// TIA Portal V17 export
// export: Created 2024-09-02T12:50:06.39653Z, ExportSetting WithDefaults, DisplayName Totally Integrated Automation Portal, DisplayVersion V17, DisplayName TIA Portal Openness, DisplayVersion V17, DisplayName TIA Portal Version Control Interface, DisplayVersion V17, DisplayName STEP 7 Professional, DisplayVersion V17, DisplayName STEP 7 Safety, DisplayVersion V17, DisplayName WinCC Professional, DisplayVersion V17
FUNCTION_BLOCK "GraFB1_FG01_Transport_OP70"   // FB1281, GRAPH
VERSION : 0.1
// stored: AcknowledgeErrorsRequired false, AutoNumber false, GraphVersion 4.0, InitialValuesAcquisition true, IsIECCheckEnabled false, LanguageInNetworks LAD, LockOperatingMode false, PermanentILProcessingInMANMode true, SetENOAutomatically false, SkipSteps false, UDAEnableTagReadback false, WithAlarmHandling true
   // inherited from GRAPH_BASE
   VAR
      OFF_SQ_BASE : Bool;
   END_VAR
   VAR_INPUT
      OFF_SQ { ExternalWritable := 'False'} : Bool := false;   // Kette ausschalten
      INIT_SQ { ExternalWritable := 'False'} : Bool := false;   // Kette in Initialzustand versetzen
      ACK_EF { ExternalWritable := 'False'} : Bool := false;   // Alle Fehler und Störungen quittieren
      S_PREV { ExternalWritable := 'False'} : Bool := false;   // Vorherigen Schritt am Parameter S_NO ausgeben
      S_NEXT { ExternalWritable := 'False'} : Bool := false;   // Nächsten Schritt am Parameter S_NO anzeigen
      SW_AUTO { ExternalWritable := 'False'} : Bool := false;   // Automtischer Betrieb
      SW_TAP { ExternalWritable := 'False'} : Bool := false;   // Halbautomatisch/Weiterschalten mit Transition
      SW_TOP { ExternalWritable := 'False'} : Bool := false;   // Halbautomatisch/Ignoriere Transition
      SW_MAN { ExternalWritable := 'False'} : Bool := false;   // Handbetrieb
      S_SEL { ExternalWritable := 'False'} : Int := 0;   // Schritt auswählen, der an S_NO ausgegeben werden soll
      S_ON { ExternalWritable := 'False'} : Bool := false;   // Schritt aktivieren, der an Parameter S_NO anliegt
      S_OFF { ExternalWritable := 'False'} : Bool := false;   // Schritt deaktivieren, der an Parameter S_NO anliegt
      T_PUSH { ExternalWritable := 'False'} : Bool := false;   // Schaltfreigabe für Transition im halbautomatischen Betrieb
   END_VAR
   VAR_OUTPUT
      S_NO { ExternalWritable := 'False'} : Int := 0;   // Schrittnummer
      S_MORE { ExternalWritable := 'False'} : Bool := false;   // Weitere Schritte sind vorhanden und können in S_NO angezeigt werden.
      S_ACTIVE { ExternalWritable := 'False'} : Bool := false;   // Schritt, der an Parameter S_NO angezeigt wird, ist aktiv
      ERR_FLT { ExternalWritable := 'False'} : Bool := false;   // Sammelfehler Interlock oder Supervision
      AUTO_ON { ExternalWritable := 'False'} : Bool := false;   // Automatischer Betrieb eingeschaltet
      TAP_ON { ExternalWritable := 'False'} : Bool := false;   // Halbautomatischer Betrieb/Schritt mit Transition eingeschaltet
      TOP_ON { ExternalWritable := 'False'} : Bool := false;   // Halbautomatischer Betrieb/Ignoriere Transition eingeschaltet
      MAN_ON { ExternalWritable := 'False'} : Bool := false;   // Handbetrieb eingeschaltet
   END_VAR
   VAR
      extBlock { S7_SetPoint := 'True'} : "LTLL_ManualGraphExt";
   END_VAR
BEGIN
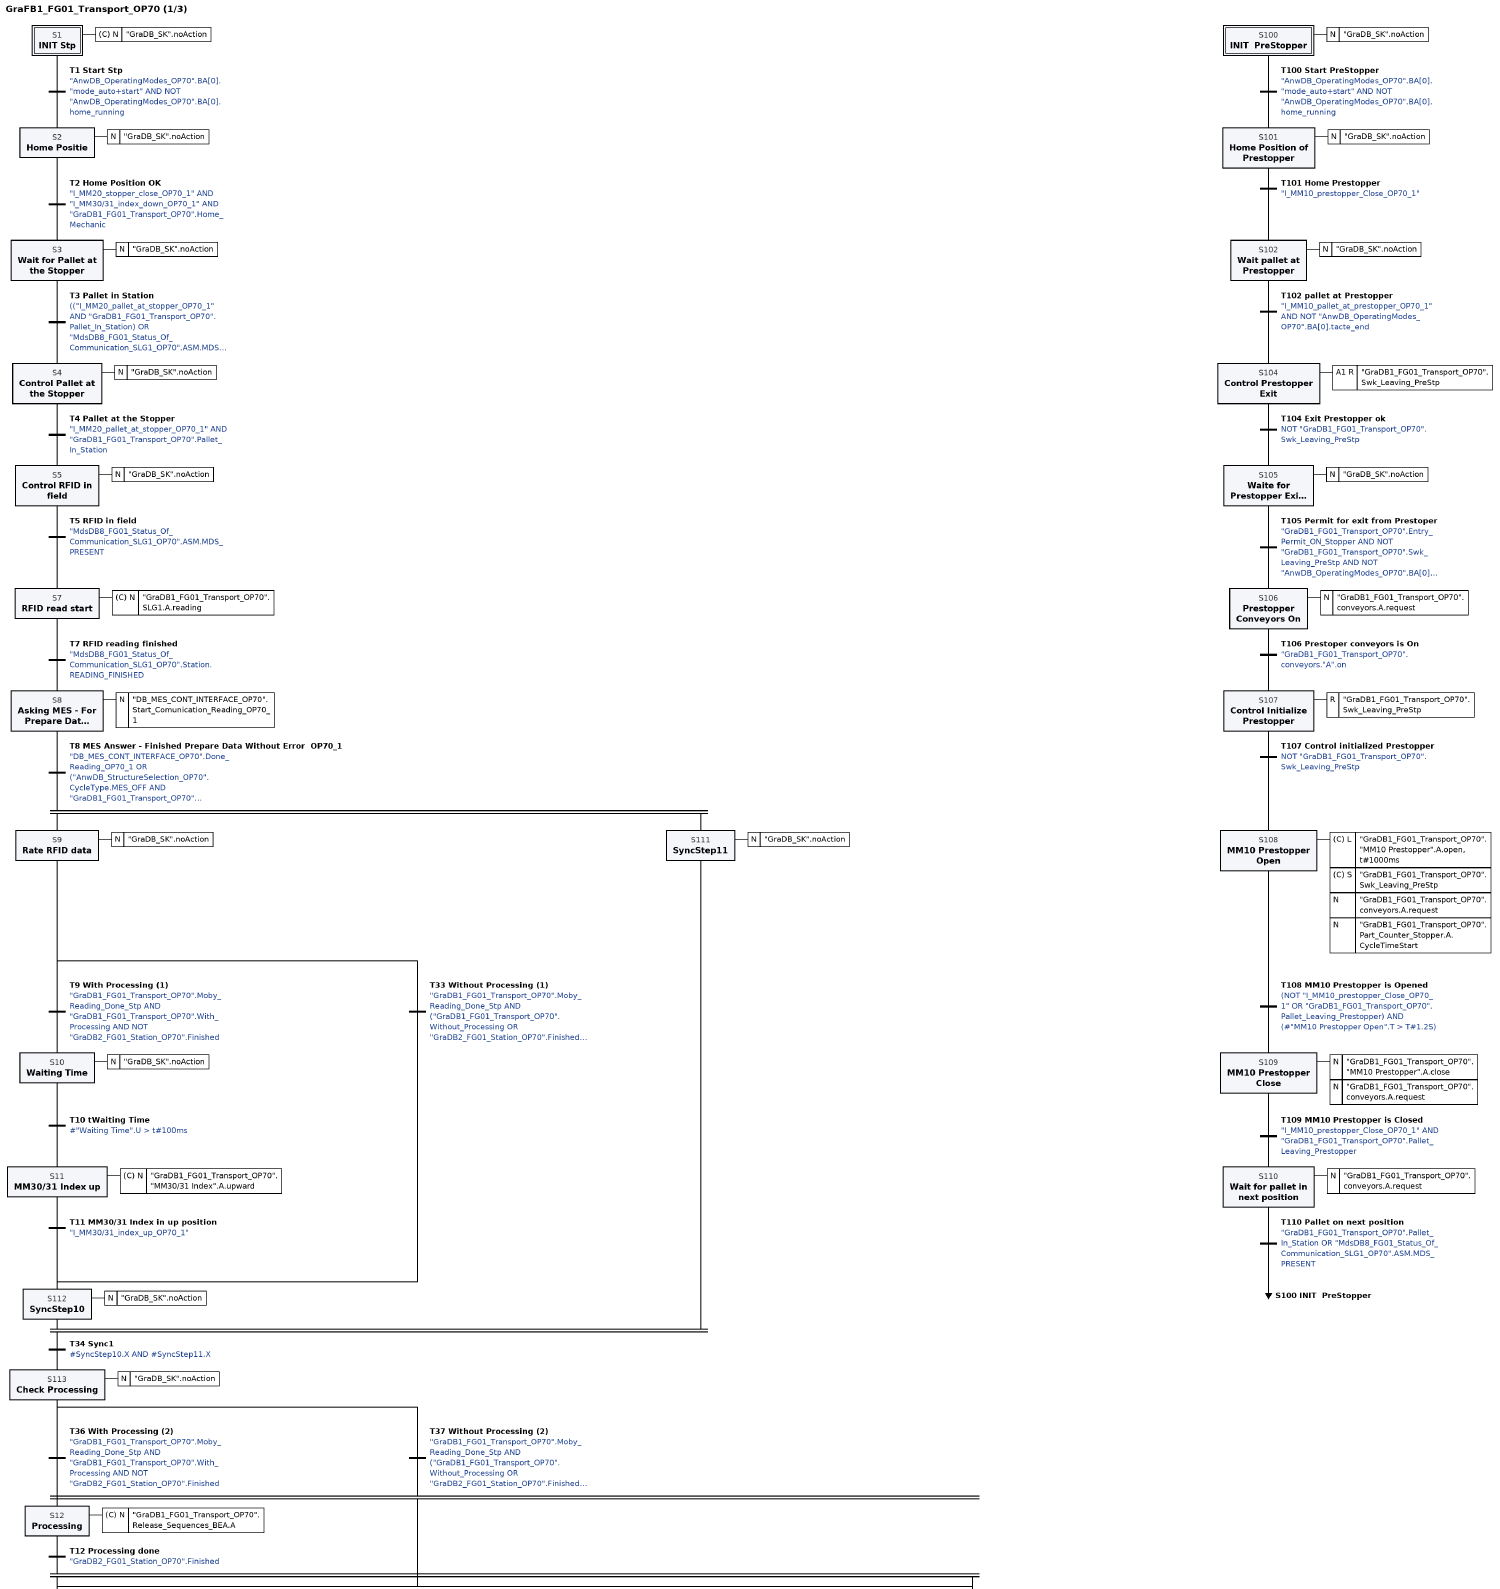
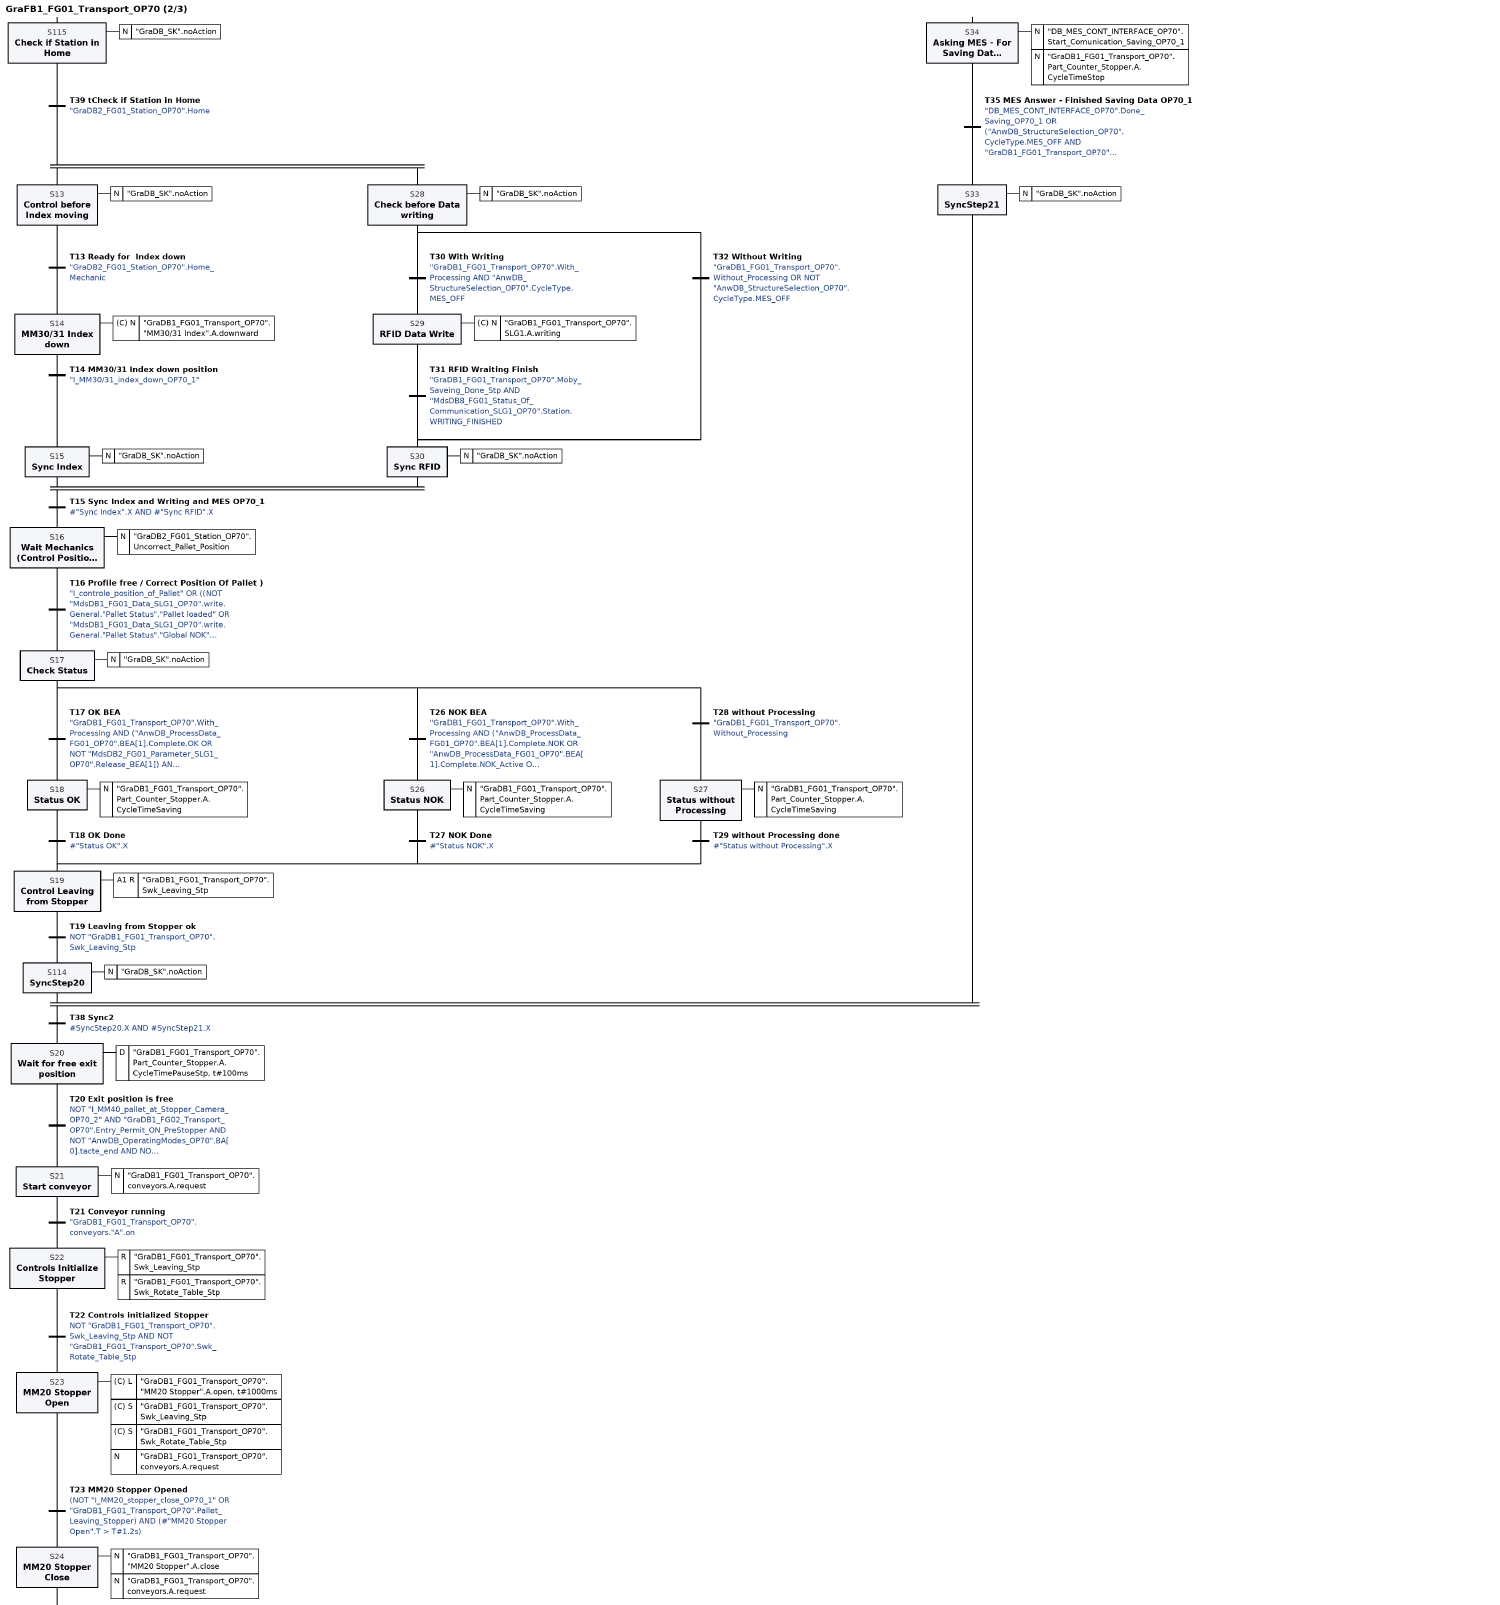
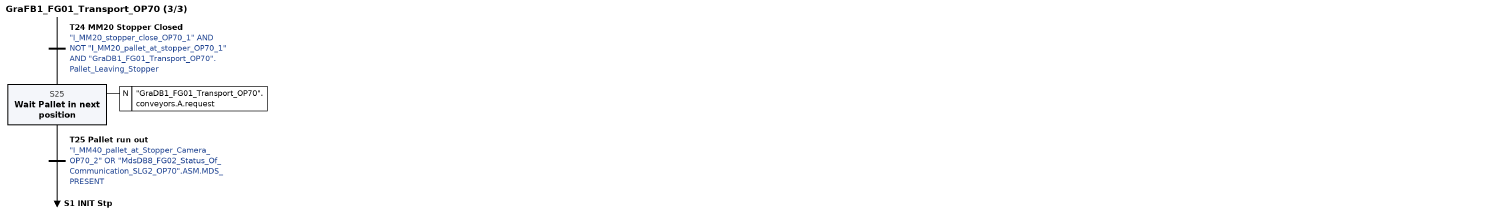
   // permanent pre-instructions
   NETWORK 1
   TITLE = HMI Lite Pass on data / HMI Lite Daten weiterreichen
      #extBlock.input := "LTLL_ManualGraphControl_OP70".screen[0].input;
   NETWORK 2
   TITLE = Instance DB Name query and pass on / Instanz DB Name abfragen und weiterreichen
      GetInstanceName(size := 0, OUT => #extBlock.input.instanceName);
   NETWORK 3
   TITLE = SK Mode
      "SysFC_SQ_Mode"(iFKT := 0, iTmsHalt := false, ioMOP := #RT_DATA.MOP);
   NETWORK 4
   TITLE = Signal change between pre-stopper and stopper / Signalwechsel Vorstopper/Stopper
      IF "GraDB1_FG01_Transport_OP70".Pallet_In_Station THEN
          "GraDB1_FG01_Transport_OP70".Swk_Leaving_PreStp := FALSE;
      END_IF;
      IF "I_MM40_pallet_at_Stopper_Camera_OP70_2" OR (NOT "GraDB1_FG01_Transport_OP70".Pallet_In_Station AND NOT "MdsDB8_FG01_Status_Of_Communication_SLG1_OP70".ASM.MDS_PRESENT AND NOT "I_MM20_pallet_at_stopper_OP70_1" AND "AlwaysFALSE") THEN
          "GraDB1_FG01_Transport_OP70".Swk_Leaving_Stp := FALSE;
      END_IF;
      IF "AlwaysTRUE" THEN "GraDB1_FG01_Transport_OP70".Swk_Rotate_Table_Stp := FALSE; END_IF;

   // sequencer 1: FG01 - Stopper MM20 / FG01 - Stopper
   INITIAL_STEP "INIT Stp":   // S1, max time T#10S, warning time T#7S
      interlock C := (none);   // Initialschritt / initial step
      supervision V := (none);   // Initialschritt / initial step
      (C)     N    "GraDB_SK".noAction
   END_STEP
   TRANSITION "Start Stp" FROM "INIT Stp" TO "Home Positie"   // T1
      := "AnwDB_OperatingModes_OP70".BA[0]."mode_auto+start" AND NOT "AnwDB_OperatingModes_OP70".BA[0].home_running;
   END_TRANSITION
   STEP "Home Positie":   // S2, max time T#10S, warning time T#7S
      supervision V := NOT #"Home Position OK".TT AND (#"Home Positie".U > T#1S);
              N    "GraDB_SK".noAction
   END_STEP
   TRANSITION "Home Position OK" FROM "Home Positie" TO "Wait for Pallet at the Stopper"   // T2
      := "I_MM20_stopper_close_OP70_1" AND "I_MM30/31_index_down_OP70_1" AND "GraDB1_FG01_Transport_OP70".Home_Mechanic;
   END_TRANSITION
   STEP "Wait for Pallet at the Stopper":   // S3, max time T#10S, warning time T#7S
              N    "GraDB_SK".noAction
   END_STEP
   TRANSITION "Pallet in Station" FROM "Wait for Pallet at the Stopper" TO "Control Pallet at the Stopper"   // T3
      := (("I_MM20_pallet_at_stopper_OP70_1" AND "GraDB1_FG01_Transport_OP70".Pallet_In_Station) OR "MdsDB8_FG01_Status_Of_Communication_SLG1_OP70".ASM.MDS_PRESENT) AND NOT "AnwDB_OperatingModes_OP70".BA[0].tacte_end;
   END_TRANSITION
   STEP "Control Pallet at the Stopper":   // S4, max time T#10S, warning time T#7S
      supervision V := NOT #"Pallet at the Stopper".TT AND (#"Control Pallet at the Stopper".U > T#5000mS);
              N    "GraDB_SK".noAction
   END_STEP
   TRANSITION "Pallet at the Stopper" FROM "Control Pallet at the Stopper" TO "Control RFID in field"   // T4
      := "I_MM20_pallet_at_stopper_OP70_1" AND "GraDB1_FG01_Transport_OP70".Pallet_In_Station;
   END_TRANSITION
   STEP "Rate RFID data":   // S9, max time T#10S, warning time T#7S
      interlock C := "MdsDB8_FG01_Status_Of_Communication_SLG1_OP70".Station.READING_FINISHED;
      supervision V := NOT #"With Processing (1)".TT AND NOT #"Without Processing (1)".TT AND (#"Rate RFID data".U > T#5000mS);
              N    "GraDB_SK".noAction
   END_STEP
   TRANSITION "With Processing (1)" FROM "Rate RFID data" TO "Waiting Time"   // T9
      := "GraDB1_FG01_Transport_OP70".Moby_Reading_Done_Stp AND "GraDB1_FG01_Transport_OP70".With_Processing AND NOT "GraDB2_FG01_Station_OP70".Finished;
   END_TRANSITION
   TRANSITION "Without Processing (1)" FROM "Rate RFID data" TO SyncStep10   // T33
      := "GraDB1_FG01_Transport_OP70".Moby_Reading_Done_Stp AND ("GraDB1_FG01_Transport_OP70".Without_Processing OR "GraDB2_FG01_Station_OP70".Finished) AND (#"Rate RFID data".T > T#500ms);
   END_TRANSITION
   STEP "MM30/31 Index up":   // S11, max time T#10S, warning time T#7S
      interlock C := "I_MM130_Press_Damper_UP_OP70_1";
      supervision V := NOT #"MM30/31 Index in up position".TT AND (#"MM30/31 Index up".U > T#5000mS);
      (C)     N    "GraDB1_FG01_Transport_OP70"."MM30/31 Index".A.upward
   END_STEP
   TRANSITION "MM30/31 Index in up position" FROM "MM30/31 Index up" TO SyncStep10   // T11
      := "I_MM30/31_index_up_OP70_1";
   END_TRANSITION
   STEP Processing:   // S12, max time T#10S, warning time T#7S
      interlock C := "MdsDB8_FG01_Status_Of_Communication_SLG1_OP70".Station.READING_FINISHED AND "I_MM30/31_index_up_OP70_1";
      (C)     N    "GraDB1_FG01_Transport_OP70".Release_Sequences_BEA.A
   END_STEP
   TRANSITION "Processing done" FROM Processing TO ("Check if Station in Home", "Asking MES - For Saving Data OP70_1")   // T12
      := "GraDB2_FG01_Station_OP70".Finished;
   END_TRANSITION
   STEP "Control before Index moving":   // S13, max time T#10S, warning time T#7S
      interlock C := "AlwaysTRUE";
      supervision V := NOT #"Ready for  Index down".TT AND (#"Control before Index moving".U > T#5000MS);
              N    "GraDB_SK".noAction
   END_STEP
   TRANSITION "Ready for  Index down" FROM "Control before Index moving" TO "MM30/31 Index  down"   // T13
      := "GraDB2_FG01_Station_OP70".Home_Mechanic;
   END_TRANSITION
   STEP "MM30/31 Index  down":   // S14, max time T#10S, warning time T#7S
      interlock C := "I_MM130_Press_Damper_UP_OP70_1";
      supervision V := NOT #"MM30/31 Index down position".TT AND (#"MM30/31 Index  down".U > T#5000mS);
      (C)     N    "GraDB1_FG01_Transport_OP70"."MM30/31 Index".A.downward
   END_STEP
   TRANSITION "MM30/31 Index down position" FROM "MM30/31 Index  down" TO "Sync Index"   // T14
      := "I_MM30/31_index_down_OP70_1";
   END_TRANSITION
   STEP "Sync Index":   // S15, max time T#10S, warning time T#7S
              N    "GraDB_SK".noAction
   END_STEP
   STEP "Check before Data writing":   // S28, max time T#10S, warning time T#7S
              N    "GraDB_SK".noAction
   END_STEP
   TRANSITION "With Writing" FROM "Check before Data writing" TO "RFID Data Write"   // T30
      := "GraDB1_FG01_Transport_OP70".With_Processing AND "AnwDB_StructureSelection_OP70".CycleType.MES_OFF;
   END_TRANSITION
   TRANSITION "Without Writing" FROM "Check before Data writing" TO "Sync RFID"   // T32
      := "GraDB1_FG01_Transport_OP70".Without_Processing OR NOT "AnwDB_StructureSelection_OP70".CycleType.MES_OFF;
   END_TRANSITION
   STEP "RFID Data Write":   // S29, max time T#10S, warning time T#7S
      interlock C := "GraDB1_FG01_Transport_OP70".Moby_Reading_Done_Stp;
      supervision V := NOT #"RFID Wraiting Finish".TT AND (#"RFID Data Write".U > T#5000MS);
      (C)     N    "GraDB1_FG01_Transport_OP70".SLG1.A.writing
   END_STEP
   TRANSITION "RFID Wraiting Finish" FROM "RFID Data Write" TO "Sync RFID"   // T31
      := "GraDB1_FG01_Transport_OP70".Moby_Saveing_Done_Stp AND "MdsDB8_FG01_Status_Of_Communication_SLG1_OP70".Station.WRITING_FINISHED;
   END_TRANSITION
   STEP "Sync RFID":   // S30, max time T#10S, warning time T#7S
              N    "GraDB_SK".noAction
   END_STEP
   TRANSITION "Sync Index and Writing and MES OP70_1" FROM ("Sync Index", "Sync RFID") TO "Wait Mechanics (Control Position Of Pallet )"   // T15
      := #"Sync Index".X AND #"Sync RFID".X;
   END_TRANSITION
   STEP "Wait Mechanics (Control Position Of Pallet )":   // S16, max time T#10S, warning time T#7S
      supervision V := NOT #"Profile free / Correct Position Of Pallet )".TT AND (#"Wait Mechanics (Control Position Of Pallet )".U > T#1000mS);
              N    "GraDB2_FG01_Station_OP70".Uncorrect_Pallet_Position
   END_STEP
   TRANSITION "Profile free / Correct Position Of Pallet )" FROM "Wait Mechanics (Control Position Of Pallet )" TO "Check Status"   // T16
      := "I_controle_position_of_Pallet" OR ((NOT "MdsDB1_FG01_Data_SLG1_OP70".write.General."Pallet Status"."Pallet loaded" OR "MdsDB1_FG01_Data_SLG1_OP70".write.General."Pallet Status"."Global NOK") AND "AnwDB_StructureSelection_OP70".CycleType.MES_OFF) OR (("DBi_Aveva_OP70_1".SettingSpecyfications.Global.General_Info.ProductStatus = 3) AND NOT "AnwDB_StructureSelection_OP70".CycleType.MES_OFF);
   END_TRANSITION
   STEP "Check Status":   // S17, max time T#10S, warning time T#7S
      supervision V := NOT #"OK BEA".TT AND NOT #"OK BEA".TT AND NOT #"without Processing".TT AND (#"Check Status".U > T#1000MS);
              N    "GraDB_SK".noAction
   END_STEP
   TRANSITION "OK BEA" FROM "Check Status" TO "Status OK"   // T17
      := "GraDB1_FG01_Transport_OP70".With_Processing AND ("AnwDB_ProcessData_FG01_OP70".BEA[1].Complete.OK OR NOT "MdsDB2_FG01_Parameter_SLG1_OP70".Release_BEA[1]) AND ("AnwDB_ProcessData_FG01_OP70".BEA[2].Complete.OK OR NOT "MdsDB2_FG01_Parameter_SLG1_OP70".Release_BEA[2]);
   END_TRANSITION
   TRANSITION "NOK BEA" FROM "Check Status" TO "Status NOK"   // T26
      := "GraDB1_FG01_Transport_OP70".With_Processing AND ("AnwDB_ProcessData_FG01_OP70".BEA[1].Complete.NOK OR "AnwDB_ProcessData_FG01_OP70".BEA[1].Complete.NOK_Active OR "AnwDB_ProcessData_FG01_OP70".BEA[2].Complete.NOK OR "AnwDB_ProcessData_FG01_OP70".BEA[2].Complete.NOK_Active);
   END_TRANSITION
   TRANSITION "without Processing" FROM "Check Status" TO "Status without Processing"   // T28
      := "GraDB1_FG01_Transport_OP70".Without_Processing;
   END_TRANSITION
   STEP "Status OK":   // S18, max time T#10S, warning time T#7S
              N    "GraDB1_FG01_Transport_OP70".Part_Counter_Stopper.A.CycleTimeSaving
   END_STEP
   TRANSITION "OK Done" FROM "Status OK" TO "Control Leaving from Stopper"   // T18
      := #"Status OK".X;
   END_TRANSITION
   STEP "Status NOK":   // S26, max time T#10S, warning time T#7S
              N    "GraDB1_FG01_Transport_OP70".Part_Counter_Stopper.A.CycleTimeSaving
   END_STEP
   TRANSITION "NOK Done" FROM "Status NOK" TO "Control Leaving from Stopper"   // T27
      := #"Status NOK".X;
   END_TRANSITION
   STEP "Status without Processing":   // S27, max time T#10S, warning time T#7S
              N    "GraDB1_FG01_Transport_OP70".Part_Counter_Stopper.A.CycleTimeSaving
   END_STEP
   TRANSITION "without Processing done" FROM "Status without Processing" TO "Control Leaving from Stopper"   // T29
      := #"Status without Processing".X;
   END_TRANSITION
   STEP "Wait for free exit position":   // S20, max time T#10S, warning time T#7S
              D    "GraDB1_FG01_Transport_OP70".Part_Counter_Stopper.A.CycleTimePauseStp, t#100ms
   END_STEP
   TRANSITION "Exit position is free" FROM "Wait for free exit position" TO "Start conveyor"   // T20
      := NOT "I_MM40_pallet_at_Stopper_Camera_OP70_2" AND "GraDB1_FG02_Transport_OP70".Entry_Permit_ON_PreStopper AND NOT "AnwDB_OperatingModes_OP70".BA[0].tacte_end AND NOT "GraDB1_FG01_Transport_OP70".Swk_Leaving_Stp AND NOT "AnwDB_OperatingModes_OP70".BA[0].tacte_end;
   END_TRANSITION
   STEP "MM20 Stopper Open":   // S23, max time T#10S, warning time T#7S
      interlock C := "I_MM30/31_index_down_OP70_1" AND NOT "I_MM40_pallet_at_Stopper_Camera_OP70_2" AND NOT "MdsDB8_FG02_Status_Of_Communication_SLG2_OP70".ASM.MDS_PRESENT AND "I_MM50_index_Camera_Down_OP70_2" AND "I_MM51_index_Camera_Down_OP70_2";
      supervision V := NOT #"MM20 Stopper Opened".TT AND (#"MM20 Stopper Open".U > T#5000mS);
      (C)     L    "GraDB1_FG01_Transport_OP70"."MM20 Stopper".A.open, t#1000ms
      (C)     S    "GraDB1_FG01_Transport_OP70".Swk_Leaving_Stp
      (C)     S    "GraDB1_FG01_Transport_OP70".Swk_Rotate_Table_Stp
              N    "GraDB1_FG01_Transport_OP70".conveyors.A.request
   END_STEP
   TRANSITION "MM20 Stopper Opened" FROM "MM20 Stopper Open" TO "MM20 Stopper Close"   // T23
      := (NOT "I_MM20_stopper_close_OP70_1" OR "GraDB1_FG01_Transport_OP70".Pallet_Leaving_Stopper) AND (#"MM20 Stopper Open".T > T#1.2s);
   END_TRANSITION
   STEP "MM20 Stopper Close":   // S24, max time T#10S, warning time T#7S
      supervision V := NOT #"MM20 Stopper Closed".TT AND (#"MM20 Stopper Close".U > T#5000mS);
              N    "GraDB1_FG01_Transport_OP70"."MM20 Stopper".A.close
              N    "GraDB1_FG01_Transport_OP70".conveyors.A.request
   END_STEP
   TRANSITION "MM20 Stopper Closed" FROM "MM20 Stopper Close" TO "Wait Pallet in next position"   // T24
      := "I_MM20_stopper_close_OP70_1" AND NOT "I_MM20_pallet_at_stopper_OP70_1" AND "GraDB1_FG01_Transport_OP70".Pallet_Leaving_Stopper;
   END_TRANSITION
   STEP "Control RFID in field":   // S5, max time T#10S, warning time T#7S
      supervision V := NOT #"RFID in field".TT AND (#"Control RFID in field".U > T#5000mS);
              N    "GraDB_SK".noAction
   END_STEP
   TRANSITION "RFID in field" FROM "Control RFID in field" TO "RFID read start"   // T5
      := "MdsDB8_FG01_Status_Of_Communication_SLG1_OP70".ASM.MDS_PRESENT;
   END_TRANSITION
   STEP "RFID read start":   // S7, max time T#10S, warning time T#7S
      interlock C := "MdsDB8_FG01_Status_Of_Communication_SLG1_OP70".ASM.MDS_PRESENT;
      supervision V := NOT #"RFID reading finished".TT AND (#"RFID read start".U > T#5000mS);
      (C)     N    "GraDB1_FG01_Transport_OP70".SLG1.A.reading
   END_STEP
   TRANSITION "RFID reading finished" FROM "RFID read start" TO "Asking MES - For Prepare Data  OP70_1"   // T7
      := "MdsDB8_FG01_Status_Of_Communication_SLG1_OP70".Station.READING_FINISHED;
   END_TRANSITION
   STEP "Start conveyor":   // S21, max time T#10S, warning time T#7S
      supervision V := NOT #"Conveyor running".TT AND (#"Start conveyor".U > T#5000MS);
              N    "GraDB1_FG01_Transport_OP70".conveyors.A.request
   END_STEP
   TRANSITION "Conveyor running" FROM "Start conveyor" TO "Controls Initialize Stopper"   // T21
      := "GraDB1_FG01_Transport_OP70".conveyors."A".on;
   END_TRANSITION
   STEP "Wait Pallet in next position":   // S25, max time T#10S, warning time T#7S
      supervision V := NOT #"Pallet run out".TT AND (#"Wait Pallet in next position".U > T#25000MS);
              N    "GraDB1_FG01_Transport_OP70".conveyors.A.request
   END_STEP
   TRANSITION "Pallet run out" FROM "Wait Pallet in next position" TO "INIT Stp"   // T25, jump
      := "I_MM40_pallet_at_Stopper_Camera_OP70_2" OR "MdsDB8_FG02_Status_Of_Communication_SLG2_OP70".ASM.MDS_PRESENT;
   END_TRANSITION
   STEP "Control Leaving from Stopper":   // S19, max time T#10S, warning time T#7S
      supervision V := NOT #"Leaving from Stopper ok".TT AND (#"Control Leaving from Stopper".U > T#1000MS);
          A1  R    "GraDB1_FG01_Transport_OP70".Swk_Leaving_Stp
   END_STEP
   TRANSITION "Leaving from Stopper ok" FROM "Control Leaving from Stopper" TO SyncStep20   // T19
      := NOT "GraDB1_FG01_Transport_OP70".Swk_Leaving_Stp;
   END_TRANSITION
   STEP "Waiting Time":   // S10, max time T#10S, warning time T#7S
      supervision V := NOT #"tWaiting Time".TT AND (#"Waiting Time".U > T#5000MS);
              N    "GraDB_SK".noAction
   END_STEP
   TRANSITION "tWaiting Time" FROM "Waiting Time" TO "MM30/31 Index up"   // T10
      := #"Waiting Time".U > t#100ms;
   END_TRANSITION
   STEP "Controls Initialize Stopper":   // S22, max time T#10S, warning time T#7S
      supervision V := NOT #"Controls initialized Stopper".TT AND (#"Controls Initialize Stopper".U > T#1000MS);
              R    "GraDB1_FG01_Transport_OP70".Swk_Leaving_Stp
              R    "GraDB1_FG01_Transport_OP70".Swk_Rotate_Table_Stp
   END_STEP
   TRANSITION "Controls initialized Stopper" FROM "Controls Initialize Stopper" TO "MM20 Stopper Open"   // T22
      := NOT "GraDB1_FG01_Transport_OP70".Swk_Leaving_Stp AND NOT "GraDB1_FG01_Transport_OP70".Swk_Rotate_Table_Stp;
   END_TRANSITION
   STEP SyncStep10:   // S112, max time T#10S, warning time T#7S
              N    "GraDB_SK".noAction
   END_STEP
   STEP SyncStep11:   // S111, max time T#10S, warning time T#7S
              N    "GraDB_SK".noAction
   END_STEP
   TRANSITION Sync1 FROM (SyncStep10, SyncStep11) TO "Check Processing"   // T34
      := #SyncStep10.X AND #SyncStep11.X;
   END_TRANSITION
   STEP "Check Processing":   // S113, max time T#10S, warning time T#7S
              N    "GraDB_SK".noAction
   END_STEP
   TRANSITION "With Processing (2)" FROM "Check Processing" TO Processing   // T36
      := "GraDB1_FG01_Transport_OP70".Moby_Reading_Done_Stp AND "GraDB1_FG01_Transport_OP70".With_Processing AND NOT "GraDB2_FG01_Station_OP70".Finished;
   END_TRANSITION
   TRANSITION "Without Processing (2)" FROM "Check Processing" TO ("Check if Station in Home", "Asking MES - For Saving Data OP70_1")   // T37
      := "GraDB1_FG01_Transport_OP70".Moby_Reading_Done_Stp AND ("GraDB1_FG01_Transport_OP70".Without_Processing OR "GraDB2_FG01_Station_OP70".Finished) AND (#"Check Processing".T > t#500ms);
   END_TRANSITION
   STEP SyncStep20:   // S114, max time T#10S, warning time T#7S
              N    "GraDB_SK".noAction
   END_STEP
   STEP "Check if Station in Home":   // S115, max time T#10S, warning time T#7S
      supervision V := NOT #"tCheck if Station in Home".TT AND (#"Check if Station in Home".U > T#3s);
              N    "GraDB_SK".noAction
   END_STEP
   TRANSITION "tCheck if Station in Home" FROM "Check if Station in Home" TO ("Control before Index moving", "Check before Data writing")   // T39
      := "GraDB2_FG01_Station_OP70".Home;
   END_TRANSITION
   STEP SyncStep21:   // S33, max time T#10S, warning time T#7S
              N    "GraDB_SK".noAction
   END_STEP
   TRANSITION Sync2 FROM (SyncStep20, SyncStep21) TO "Wait for free exit position"   // T38
      := #SyncStep20.X AND #SyncStep21.X;
   END_TRANSITION
   STEP "Asking MES - For Saving Data OP70_1":   // S34, max time T#10S, warning time T#7S
      interlock C := "MdsDB8_FG01_Status_Of_Communication_SLG1_OP70".ASM.MDS_PRESENT OR 1;
      supervision V := NOT #"MES Answer - Finished Saving Data OP70_1".TT AND (#"Asking MES - For Saving Data OP70_1".U > T#5s) AND 0;
              N    "DB_MES_CONT_INTERFACE_OP70".Start_Comunication_Saving_OP70_1
              N    "GraDB1_FG01_Transport_OP70".Part_Counter_Stopper.A.CycleTimeStop
   END_STEP
   TRANSITION "MES Answer - Finished Saving Data OP70_1" FROM "Asking MES - For Saving Data OP70_1" TO SyncStep21   // T35
      := "DB_MES_CONT_INTERFACE_OP70".Done_Saving_OP70_1 OR ("AnwDB_StructureSelection_OP70".CycleType.MES_OFF AND "GraDB1_FG01_Transport_OP70".Tracebility_off) OR "AnwDB_StructureSelection_OP70".UserDefine.IbmMode;
   END_TRANSITION
   STEP "Asking MES - For Prepare Data  OP70_1":   // S8, max time T#10S, warning time T#7S
      interlock C := "MdsDB8_FG01_Status_Of_Communication_SLG1_OP70".ASM.MDS_PRESENT OR 1;
      supervision V := NOT #"MES Answer - Finished Prepare Data Without Error  OP70_1".TT AND (#"Asking MES - For Prepare Data  OP70_1".U > T#7s);
              N    "DB_MES_CONT_INTERFACE_OP70".Start_Comunication_Reading_OP70_1
   END_STEP
   TRANSITION "MES Answer - Finished Prepare Data Without Error  OP70_1" FROM "Asking MES - For Prepare Data  OP70_1" TO ("Rate RFID data", SyncStep11)   // T8
      := "DB_MES_CONT_INTERFACE_OP70".Done_Reading_OP70_1 OR ("AnwDB_StructureSelection_OP70".CycleType.MES_OFF AND "GraDB1_FG01_Transport_OP70".Tracebility_off) OR "AnwDB_StructureSelection_OP70".UserDefine.IbmMode;
   END_TRANSITION

   // sequencer 2: FG01 - PreStopper MM10 / FG01 - Vorstopper
   INITIAL_STEP "INIT  PreStopper":   // S100, max time T#10S, warning time T#7S: Activate if pre-stop is available / Aktivieren, wenn Vorstopper vorhanden
              N    "GraDB_SK".noAction
   END_STEP
   TRANSITION "Start PreStopper" FROM "INIT  PreStopper" TO "Home Position of Prestopper"   // T100
      := "AnwDB_OperatingModes_OP70".BA[0]."mode_auto+start" AND NOT "AnwDB_OperatingModes_OP70".BA[0].home_running;
   END_TRANSITION
   STEP "Home Position of Prestopper":   // S101, max time T#10S, warning time T#7S
      supervision V := NOT #"Home Prestopper".TT AND (#"Home Position of Prestopper".U > T#1S);
              N    "GraDB_SK".noAction
   END_STEP
   TRANSITION "Home Prestopper" FROM "Home Position of Prestopper" TO "Wait pallet at Prestopper"   // T101
      := "I_MM10_prestopper_Close_OP70_1";
   END_TRANSITION
   STEP "Wait pallet at Prestopper":   // S102, max time T#10S, warning time T#7S
              N    "GraDB_SK".noAction
   END_STEP
   TRANSITION "pallet at Prestopper" FROM "Wait pallet at Prestopper" TO "Control Prestopper Exit"   // T102
      := "I_MM10_pallet_at_prestopper_OP70_1" AND NOT "AnwDB_OperatingModes_OP70".BA[0].tacte_end;
   END_TRANSITION
   STEP "MM10 Prestopper Open":   // S108, max time T#10S, warning time T#7S
      interlock C := NOT "I_MM20_pallet_at_stopper_OP70_1" AND NOT "MdsDB8_FG01_Status_Of_Communication_SLG1_OP70".ASM.MDS_PRESENT AND "I_MM30/31_index_down_OP70_1" AND "I_MM130_Press_Damper_UP_OP70_1";
      supervision V := NOT #"MM10 Prestopper is Opened".TT AND (#"MM10 Prestopper Open".U > T#5000MS);
      (C)     L    "GraDB1_FG01_Transport_OP70"."MM10 Prestopper".A.open, t#1000ms
      (C)     S    "GraDB1_FG01_Transport_OP70".Swk_Leaving_PreStp
              N    "GraDB1_FG01_Transport_OP70".conveyors.A.request
              N    "GraDB1_FG01_Transport_OP70".Part_Counter_Stopper.A.CycleTimeStart
   END_STEP
   TRANSITION "MM10 Prestopper is Opened" FROM "MM10 Prestopper Open" TO "MM10 Prestopper Close"   // T108
      := (NOT "I_MM10_prestopper_Close_OP70_1" OR "GraDB1_FG01_Transport_OP70".Pallet_Leaving_Prestopper) AND (#"MM10 Prestopper Open".T > T#1.2S);
   END_TRANSITION
   STEP "MM10 Prestopper Close":   // S109, max time T#10S, warning time T#7S
      supervision V := NOT #"MM10 Prestopper is Closed".TT AND (#"MM10 Prestopper Close".U > T#5000MS);
              N    "GraDB1_FG01_Transport_OP70"."MM10 Prestopper".A.close
              N    "GraDB1_FG01_Transport_OP70".conveyors.A.request
   END_STEP
   TRANSITION "MM10 Prestopper is Closed" FROM "MM10 Prestopper Close" TO "Wait for pallet in next position"   // T109
      := "I_MM10_prestopper_Close_OP70_1" AND "GraDB1_FG01_Transport_OP70".Pallet_Leaving_Prestopper;
   END_TRANSITION
   STEP "Waite for Prestopper Exit Free":   // S105, max time T#10S, warning time T#7S
              N    "GraDB_SK".noAction
   END_STEP
   TRANSITION "Permit for exit from Prestoper" FROM "Waite for Prestopper Exit Free" TO "Prestopper Conveyors On"   // T105
      := "GraDB1_FG01_Transport_OP70".Entry_Permit_ON_Stopper AND NOT "GraDB1_FG01_Transport_OP70".Swk_Leaving_PreStp AND NOT "AnwDB_OperatingModes_OP70".BA[0].tacte_end;
   END_TRANSITION
   STEP "Wait for pallet in next position":   // S110, max time T#10S, warning time T#7S
      supervision V := NOT #"Pallet on next position".TT AND (#"Wait for pallet in next position".U > T#15000MS);
              N    "GraDB1_FG01_Transport_OP70".conveyors.A.request
   END_STEP
   TRANSITION "Pallet on next position" FROM "Wait for pallet in next position" TO "INIT  PreStopper"   // T110, jump
      := "GraDB1_FG01_Transport_OP70".Pallet_In_Station OR "MdsDB8_FG01_Status_Of_Communication_SLG1_OP70".ASM.MDS_PRESENT;
   END_TRANSITION
   STEP "Prestopper Conveyors On":   // S106, max time T#10S, warning time T#7S
      supervision V := NOT #"Prestoper conveyors is On".TT AND (#"Prestopper Conveyors On".U > T#5000MS);
              N    "GraDB1_FG01_Transport_OP70".conveyors.A.request
   END_STEP
   TRANSITION "Prestoper conveyors is On" FROM "Prestopper Conveyors On" TO "Control Initialize Prestopper"   // T106
      := "GraDB1_FG01_Transport_OP70".conveyors."A".on;
   END_TRANSITION
   STEP "Control Prestopper Exit":   // S104, max time T#10S, warning time T#7S
      supervision V := NOT #"Exit Prestopper ok".TT AND (#"Control Prestopper Exit".U > T#1000MS);
          A1  R    "GraDB1_FG01_Transport_OP70".Swk_Leaving_PreStp
   END_STEP
   TRANSITION "Exit Prestopper ok" FROM "Control Prestopper Exit" TO "Waite for Prestopper Exit Free"   // T104
      := NOT "GraDB1_FG01_Transport_OP70".Swk_Leaving_PreStp;
   END_TRANSITION
   STEP "Control Initialize Prestopper":   // S107, max time T#10S, warning time T#7S
      supervision V := NOT #"Control initialized Prestopper".TT AND (#"Control Initialize Prestopper".U > T#1000MS);
              R    "GraDB1_FG01_Transport_OP70".Swk_Leaving_PreStp
   END_STEP
   TRANSITION "Control initialized Prestopper" FROM "Control Initialize Prestopper" TO "MM10 Prestopper Open"   // T107
      := NOT "GraDB1_FG01_Transport_OP70".Swk_Leaving_PreStp;
   END_TRANSITION

   // permanent post-instructions
   NETWORK 1
   TITLE = Move interlocks from Ext block to ManualGraphControl DB / Interlocks vom Ext-Block zum ManualGraphControl DB rangieren
      "LTLL_ManualGraphInterlock"(ManualGraphExtOutput := #extBlock.output,
                              ManualGraphControlScreen := "LTLL_ManualGraphControl_OP70".screen[0]);
   NETWORK 2
   TITLE = Report step error / Schrittkettenfehler melden
      "SysFC_NumOfSQErrors"(FLT := #RT_DATA.SQ_FLAGS.ERR_FLT,
                            Fault_SQ := "AnwDB_OperatingModes_OP70".BA[0].error_report_SK,
                            NumOf_Fault_SQ := "AnwDB_ZP_Alarm_OP70".FaultsNoSK_ST1);
   NETWORK 3
   TITLE = Basic position Step chain / Grundstellung Schrittkette
      "GraDB1_FG01_Transport_OP70".Home_SQ := (#"INIT  PreStopper".X OR #"Wait pallet at Prestopper".X OR #"Waite for Prestopper Exit Free".X) AND (#"INIT Stp".X OR #"Wait for Pallet at the Stopper".X OR #"Wait for free exit position".X);
   NETWORK 4
   TITLE = WT is run out Vorstopper / Stopper / WT ist Ausgelaufen Vorstopper / Stopper
      "GraDB1_FG01_Transport_OP70".Pallet_Leaving_Prestopper := (#"MM10 Prestopper Open".X OR #"MM10 Prestopper Close".X) AND (NOT "I_MM10_pallet_at_prestopper_OP70_1" OR "GraDB1_FG01_Transport_OP70".Pallet_Leaving_Prestopper);
      "GraDB1_FG01_Transport_OP70".Pallet_Leaving_Stopper := (#"MM20 Stopper Open".X OR #"MM20 Stopper Close".X) AND ((NOT "I_MM20_pallet_at_stopper_OP70_1" AND NOT "MdsDB8_FG01_Status_Of_Communication_SLG1_OP70".ASM.MDS_PRESENT) OR "GraDB1_FG01_Transport_OP70".Pallet_Leaving_Stopper);
   NETWORK 5
   TITLE = Enable inlet / Freigabe Einlauf
      "GraDB1_FG01_Transport_OP70".Entry_Permit_ON_Stopper := ((#"Wait for Pallet at the Stopper".X AND NOT "MdsDB8_FG01_Status_Of_Communication_SLG1_OP70".ASM.MDS_PRESENT AND NOT "I_MM20_pallet_at_stopper_OP70_1") OR (#"MM20 Stopper Open".X AND NOT #"MM20 Stopper Open".LA AND "AlwaysFALSE") OR #"MM20 Stopper Close".X) AND "GraDB1_FG01_Transport_OP70".Home_Mechanic AND "I_MM30/31_index_down_OP70_1" AND "I_MM130_Press_Damper_UP_OP70_1";
   NETWORK 6
   TITLE = Wait for WT / Warte auf WT
      "GraDB1_FG01_Transport_OP70".Wait_For_Pallet := (#"Wait pallet at Prestopper".X OR #"INIT  PreStopper".X) AND #"Wait for Pallet at the Stopper".X;
END_FUNCTION_BLOCK
